FUNCTION_BLOCK FB_Sum_Test EXTENDS TcUnit.FB_TestSuite
VAR
END_VAR

TwoPlusTwoEqualsFour();
ZeroPlusZeroEqualsZero();

METHOD PRIVATE TwoPlusTwoEqualsFour
VAR
	Sum : FB_Sum;
	Result : UINT;
    ExpectedSum : UINT := 4;
END_VAR
TEST('TwoPlusTwoEqualsFour');

Sum(one := 2, two := 2, result => Result);

AssertEquals(Expected := ExpectedSum,
             Actual := Result,
             Message := 'The calculation is not correct');

TEST_FINISHED();
END_METHOD

METHOD PRIVATE ZeroPlusZeroEqualsZero
VAR
	Sum : FB_Sum;
	Result : UINT;
    ExpectedSum : UINT := 0;
END_VAR
TEST('ZeroPlusZeroEqualsZero');

Sum(one := 0, two := 0, result => Result);

AssertEquals(Expected := ExpectedSum,
             Actual := Result,
             Message := 'The calculation is not correct');

TEST_FINISHED();
END_METHOD

END_FUNCTION_BLOCK

(* stored: Version 1.1.0.1, ProductVersion 3.1.4022.18
   POU FB_Sum_Test: Id {69b661ca-5faa-43bb-8b8a-2cae13b2cfe4}, SpecialFunc None
   Method TwoPlusTwoEqualsFour: Id {071ba4c3-fe0d-4b0b-be72-a320c9d403a4}
   Method ZeroPlusZeroEqualsZero: Id {ac47aa92-0e7a-4876-b0ac-7ef29219d372} *)
